{attribute 'qualified_only'}
//{attribute 'strict'}
{attribute 'to_string'}
TYPE E_JOB_STATE :
(
	JOB_NULL,
  JOB_INIT    := 10,
  JOB_IDLE,
  JOB_RESET,
  JOB_HOME,
  JOB_RINSE,
  JOB_AUTO    := 20
)UINT;
END_TYPE

(* stored: Version 1.1.0.1
   DUT E_JOB_STATE: Id {84de87e5-18f8-4d91-9c74-5298dd0bfeea} *)
